PROGRAM DNS_SNTP_SYSLOG_DEMO
VAR
	IP_C : IP_C;
	S_BUF : NETWORK_BUFFER;
	R_BUF : NETWORK_BUFFER;
	IP_CONTROL_1: IP_CONTROL;
	DNS_CLIENT : DNS_CLIENT;
	SNTP_CLIENT: SNTP_CLIENT;
	SNTP_SERVER: SNTP_SERVER;
	COUNT_DR: COUNT_DR;
	RTC_2: RTC_2;
	count_cycles: DWORD;
	dns_error: DWORD;
	sntp_error: DWORD;
	freigabe: BOOL;
	dso: BOOL;
	xms: INT;
	sntp_srv_enable: BOOL;
	cur_UDT: DT;
	cur_LDT: DT;
	SYS_LOG: SYS_LOG;
	sys_log_option: BYTE := 2#0000_0100;
	TON_1: TON;
	tp_sys_log: BOOL;
	error_sys_log: DWORD;
	sys_time: TIME;
END_VAR
VAR // added by the converter: edge detectors and wires of the graphical bodies
    _w1, _w2 : ANY;
END_VAR

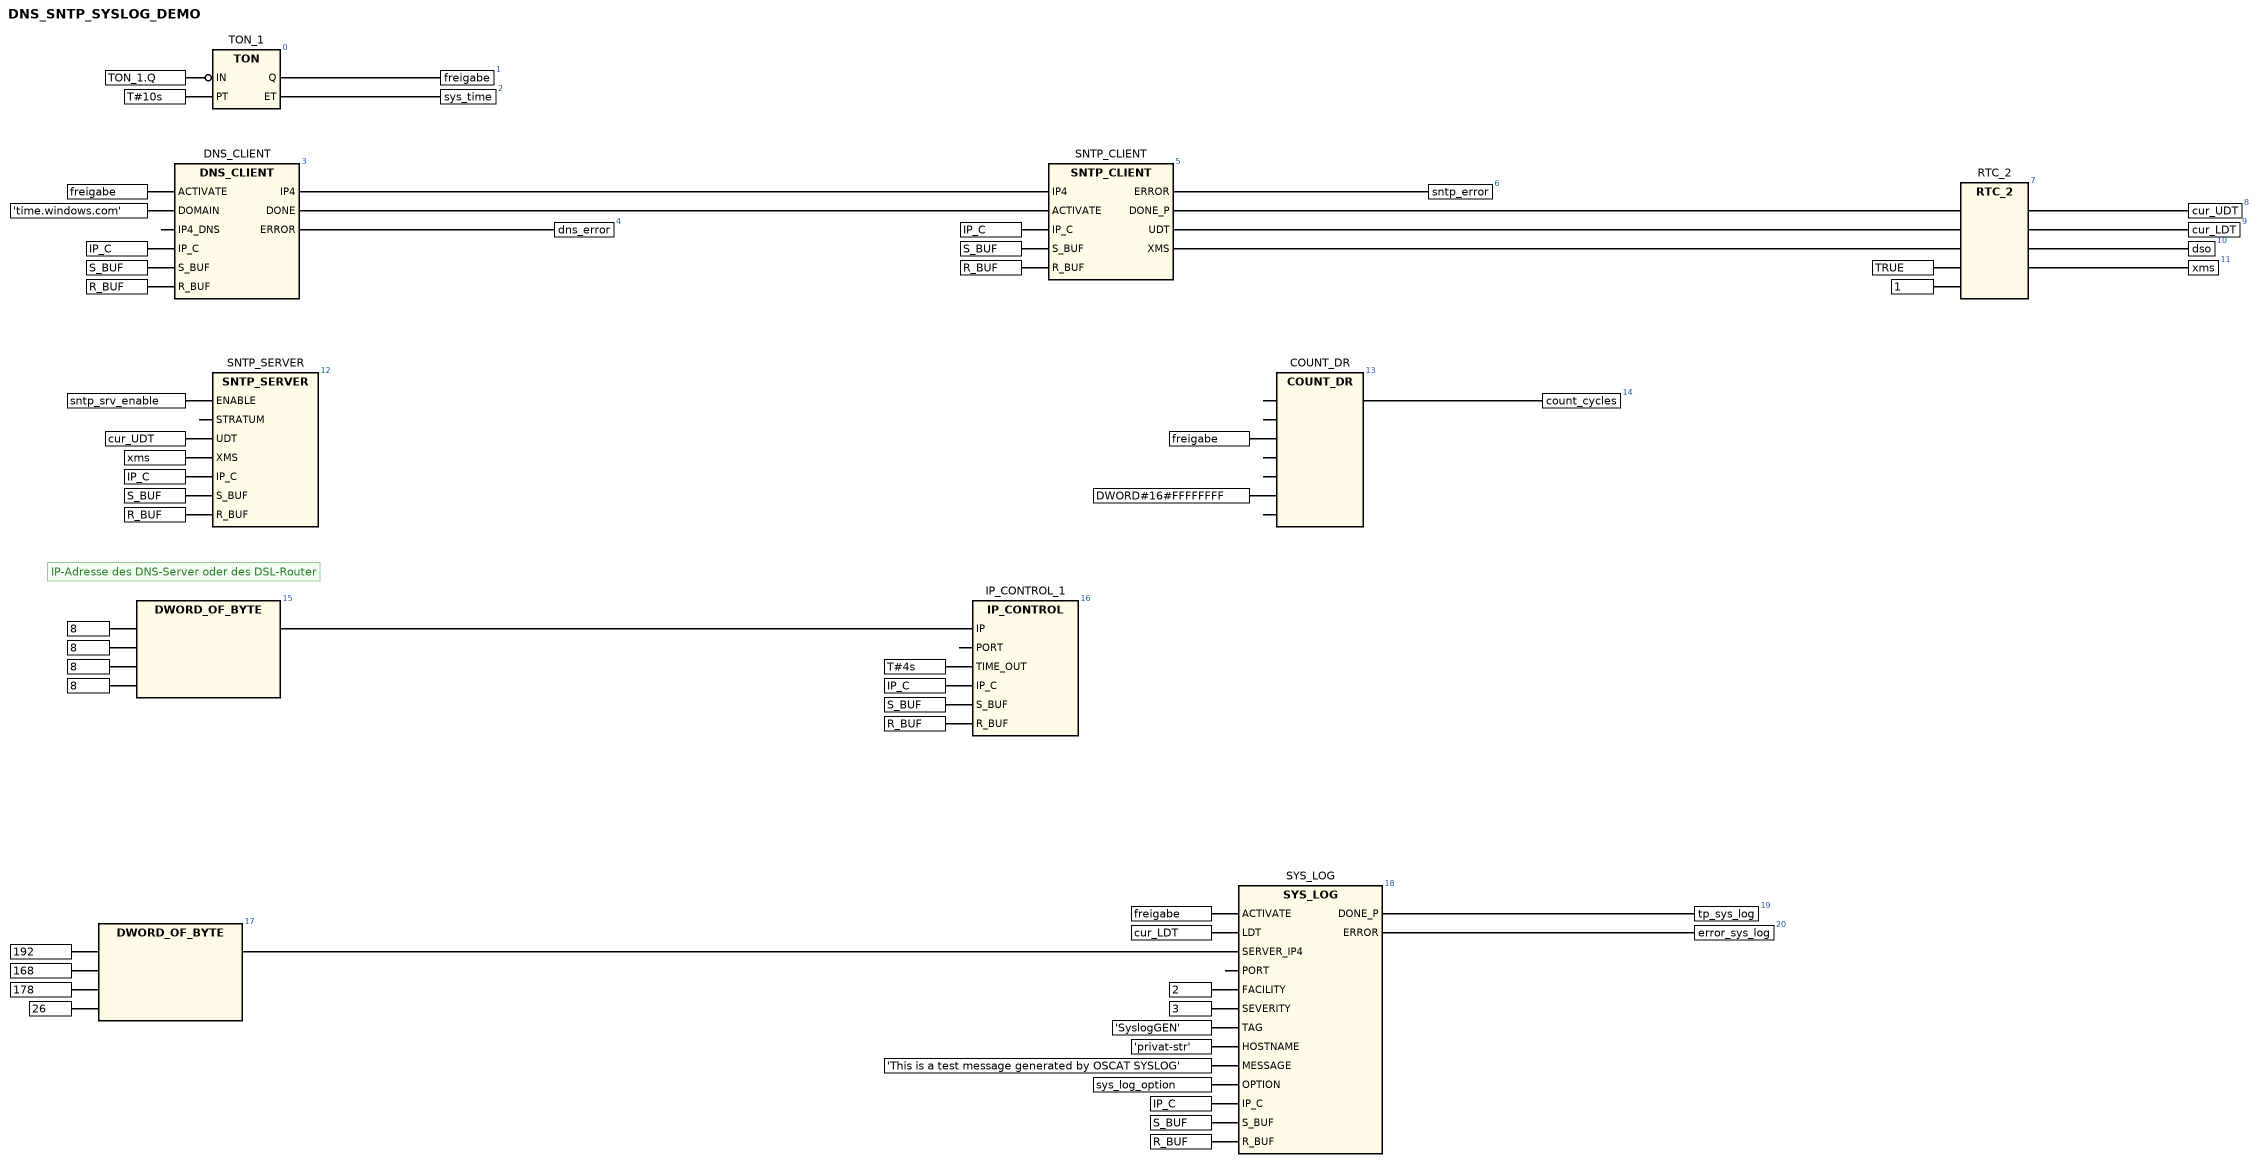
TON_1(IN := NOT TON_1.Q, PT := T#10s); // TON
freigabe := TON_1.Q;
sys_time := TON_1.ET;
DNS_CLIENT(ACTIVATE := freigabe, DOMAIN := 'time.windows.com', IP_C := IP_C, S_BUF := S_BUF, R_BUF := R_BUF);
dns_error := DNS_CLIENT.ERROR;
SNTP_CLIENT(IP4 := DNS_CLIENT.IP4, ACTIVATE := DNS_CLIENT.DONE, IP_C := IP_C, S_BUF := S_BUF, R_BUF := R_BUF);
sntp_error := SNTP_CLIENT.ERROR;
RTC_2(_in1 := SNTP_CLIENT.DONE_P, _in2 := SNTP_CLIENT.UDT, _in3 := SNTP_CLIENT.XMS, _in4 := TRUE, _in5 := 1);
cur_UDT := RTC_2._out1;
cur_LDT := RTC_2._out2;
dso := RTC_2._out3;
xms := RTC_2._out4;
SNTP_SERVER(
    ENABLE := sntp_srv_enable,
    UDT := cur_UDT,
    XMS := xms,
    IP_C := IP_C,
    S_BUF := S_BUF,
    R_BUF := R_BUF);
COUNT_DR(_in3 := freigabe, _in6 := DWORD#16#FFFFFFFF);
count_cycles := COUNT_DR._out1;
// IP-Adresse des DNS-Server oder des DSL-Router
_w1 := DWORD_OF_BYTE(8, 8, 8, 8);
IP_CONTROL_1(IP := _w1, TIME_OUT := T#4s, IP_C := IP_C, S_BUF := S_BUF, R_BUF := R_BUF); // IP_CONTROL
_w2 := DWORD_OF_BYTE(192, 168, 178, 26);
SYS_LOG(
    ACTIVATE := freigabe,
    LDT := cur_LDT,
    SERVER_IP4 := _w2,
    FACILITY := 2,
    SEVERITY := 3,
    TAG := 'SyslogGEN',
    HOSTNAME := 'privat-str',
    MESSAGE := 'This is a test message generated by OSCAT SYSLOG',
    OPTION := sys_log_option,
    IP_C := IP_C,
    S_BUF := S_BUF,
    R_BUF := R_BUF);
tp_sys_log := SYS_LOG.DONE_P;
error_sys_log := SYS_LOG.ERROR;

END_PROGRAM

(* stored: Version 1.1.0.1, ProductVersion 3.1.4024.9
   POU DNS_SNTP_SYSLOG_DEMO: Id {b6f934b2-982d-42af-a9ab-4bf5fdb0daae}, SpecialFunc None *)
